(* PLC project Unnamed, 不明 Unnamed 1 *)
(* stored: creationDateTime 2025-07-18T14:58:35, modificationDateTime 2025-08-10T16:01:33 *)

CONFIGURATION Config0
  RESOURCE Res0 ON PLC
  END_RESOURCE
END_CONFIGURATION
